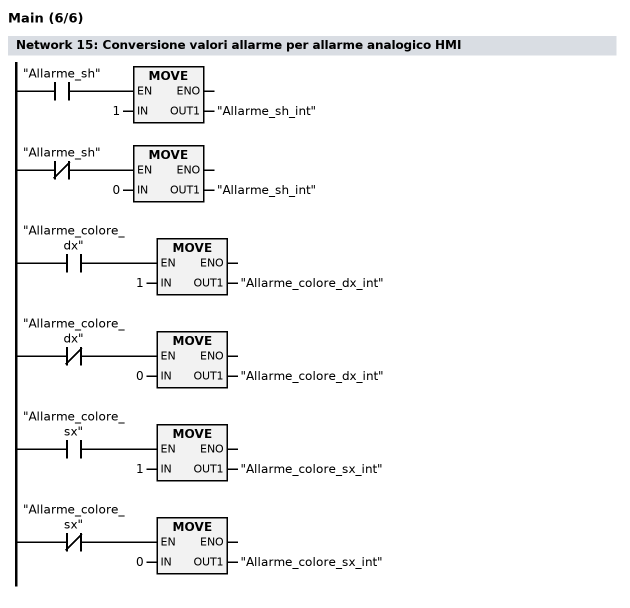
   RUNG wire#powerrail
      Contact( "Allarme_sh" )
      Move(in := 1, out1 => "Allarme_sh_int")
   END_RUNG
   RUNG wire#powerrail
      I_Contact( "Allarme_sh" )
      Move(in := 0, out1 => "Allarme_sh_int")
   END_RUNG
   RUNG wire#powerrail
      Contact( "Allarme_colore_dx" )
      Move(in := 1, out1 => "Allarme_colore_dx_int")
   END_RUNG
   RUNG wire#powerrail
      I_Contact( "Allarme_colore_dx" )
      Move(in := 0, out1 => "Allarme_colore_dx_int")
   END_RUNG
   RUNG wire#powerrail
      Contact( "Allarme_colore_sx" )
      Move(in := 1, out1 => "Allarme_colore_sx_int")
   END_RUNG
   RUNG wire#powerrail
      I_Contact( "Allarme_colore_sx" )
      Move(in := 0, out1 => "Allarme_colore_sx_int")
   END_RUNG
   // the same network as SCL:
   IF "Allarme_sh" THEN "Allarme_sh_int" := 1; END_IF;
   IF NOT "Allarme_sh" THEN "Allarme_sh_int" := 0; END_IF;
   IF "Allarme_colore_dx" THEN "Allarme_colore_dx_int" := 1; END_IF;
   IF NOT "Allarme_colore_dx" THEN "Allarme_colore_dx_int" := 0; END_IF;
   IF "Allarme_colore_sx" THEN "Allarme_colore_sx_int" := 1; END_IF;
   IF NOT "Allarme_colore_sx" THEN "Allarme_colore_sx_int" := 0; END_IF;
END_REGION
END_ORGANIZATION_BLOCK

(* ===== HMI "HMI_RT_1" =====
system functions are stored by id; their names below are inferred from use
connection "HMI_Connection_1": ETHERNET, SMART_S7_1200_OMS

HMI tags "Default tag table"
   "HMI_Robot" : Bool = PLC "Pick-place_DB".work AT %Q0.1, 1 s
   "HMI_ElevatorDx" : Bool = PLC Elevator_dx_DB.pronto_ricevere AT %I1.5, 1 s
   "HMI_ElevatorSx" : Bool = PLC Elevator_sx_DB.pronto_ricevere AT %I1.6, 1 s
   "HMI_Impianto" : Bool = PLC Impianto_attivo AT %M0.0, 1 s
   "HMI_Start" : Bool = PLC Cmd_start AT %M0.1, 1 s
   "HMI_Stop" : Bool = PLC Cmd_stop AT %M0.2, 1 s
   "HMI_Totali" : Int = PLC Pezzi_totali AT %MW10, 1 s
   "HMI_Blu" : Int = PLC Pezzi_blu AT %MW12, 1 s
   "HMI_Verdi" : Int = PLC Pezzi_verdi AT %MW14, 1 s
   "HMI_Grigi" : Int = PLC Pezzi_grigi AT %MW16, 1 s
   "HMI_Sospendi" : Bool = PLC Sospendi AT %M0.5, 1 s
   "HMI_Reset" : Bool = PLC Reset AT %M0.4, 1 s
   "HMI_Stato_sospeso" : Bool = PLC Supervisore_DB.Stato_sospeso AT %DB1.DBW0, 1 s
   "HMI_Stato_allarme_attivo" : Bool = PLC Allarme AT %M0.3, 1 s
   "Allarme_sh" : Bool = PLC Allarme_sh AT %M1.0, 1 s
   "Allarme_colore_sx" : Bool = PLC Allarme_colore_sx AT %M0.7, 1 s
   "Allarme_colore_dx" : Bool = PLC Allarme_colore_dx AT %M0.6, 1 s
   "HMI_Allarme_sh_int" : Int = PLC Allarme_sh_int AT %MW20, 1 s
   "HMI_Allarme_colore_dx_int" : Int = PLC Allarme_colore_dx_int AT %MW22, 1 s
   "HMI_Allarme_colore_sx_int" : Int = PLC Allarme_colore_sx_int AT %MW24, 1 s

analog alarms
   1: 'ALLARME: pezzo mancante dopo il robot', class Errors, trigger "HMI_Allarme_sh_int"
   2: 'ALLARME: colore non rilevato sul nastro destro', class Errors, trigger "HMI_Allarme_colore_dx_int"
   3: 'ALLARME: colore non rilevato sul nastro sinistro', class Errors, trigger "HMI_Allarme_colore_sx_int"

screen "Home" 800x480, template "Template_1"
   Button "HmiScreenItemData" at 7,42 size 173x59; TextOn 'Forzature'; TextOff 'Supervisione impianto'; PictureOn "Navigates to Forzature for KTP900 Basic+ PN 17.0.0.0"; PictureOff "Navigates to Forzature for KTP900 Basic+ PN 17.0.0.0"
      on Click: ActivateScreen("Supervisione impianto", 0)
   TextField "Text field_1" at 28,104 size 286x27; Text 'STATO GENERALE IMPIANTO'
   TextField "Text field_2" at 563,104 size 187x27; Text 'CONTEGGIO PEZZI'
   TextField "Text field_3" at 362,103 size 101x27; Text 'COMANDI'
   TextField "Text field_5" at 198,53 size 546x25; Text 'IMPIANTO DI PRODUZIONE E SMISTAMENTO AUTOMATIZZATO'
   TextField "Text field_6" at 562,158 size 68x25; Text 'TOTALI'
   TextField "Text field_7" at 568,215 size 40x25; Text 'BLU'
   TextField "Text field_8" at 562,269 size 59x25; Text 'VERDI'
   TextField "Text field_9" at 562,329 size 59x25; Text 'GRIGI'
   TextField "Text field_13" at 45,210 size 101x20; Text 'ROBOT PRONTO'
   TextField "Text field_15" at 21,268 size 177x20; Text 'ELEVATOR DESTRO PRONTO'
   TextField "Text field_14" at 19,332 size 187x20; Text 'ELEVATOR SINISTRO PRONTO'
   Circle "Circle_2" at 228,199 size 43x43
      Appearance <- "HMI_Robot"
   Circle "Circle_3" at 229,257 size 44x44
      Appearance <- "HMI_ElevatorDx"
   Circle "Circle_4" at 228,323 size 45x45
      Appearance <- "HMI_ElevatorSx"
   IOField "I/O field_1" at 654,154 size 96x32; FormatPattern s99999
      ProcessValue <- "HMI_Totali"
   IOField "I/O field_2" at 654,210 size 96x32; FormatPattern s99999
      ProcessValue <- "HMI_Blu"
   IOField "I/O field_3" at 656,266 size 96x32; FormatPattern s99999
      ProcessValue <- "HMI_Verdi"
   IOField "I/O field_4" at 654,329 size 96x32; FormatPattern s99999
      ProcessValue <- "HMI_Grigi"
   Button "Button_2" at 357,249 size 120x71; TextOff 'ARRESTO'
      on Release: ResetBit("HMI_Stop")
      on Press: SetBit("HMI_Stop")
   Button "Button_3" at 357,162 size 119x63; TextOff 'AVVIO'
      on Release: ResetBit("HMI_Start")
      on Press: SetBit("HMI_Start")
   TextField "Text field_4" at 50,154 size 119x20; Text 'IMPIANTO ATTIVO'
   Circle "Circle_1" at 226,141 size 42x42
      Appearance <- "HMI_Impianto"

screen "Supervisione impianto" 800x480, template "Template_1"
   TextField "HmiScreenItemData" at 157,55 size 505x33; Text 'Supervisione impianto'
   Button "Back" at 1,41 size 159x47; TextOn 'Back'; TextOff 'Home'
      on Click: ActivateScreen("Home", 0)
   Button "Button_1" at 54,139 size 163x69; TextOff 'SOSPENDI'
      on Press: SetBit("HMI_Sospendi")
      on Release: ResetBit("HMI_Sospendi")
   Button "Button_2" at 58,243 size 158x71; TextOff 'RESET'
      on Press: SetBit("HMI_Reset")
      on Release: ResetBit("HMI_Reset")
   TextField "Text field_1" at 260,157 size 165x27; Text 'STATO SOSPESO'
   Circle "Circle_1" at 471,145 size 48x48
      Appearance <- "HMI_Stato_sospeso"
   TextField "Text field_2" at 261,261 size 176x27; Text 'ALLARME ATTIVO'
   Circle "Circle_2" at 471,248 size 48x48
      Appearance <- "HMI_Stato_allarme_attivo"
   TextField "Text field_4" at 583,100 size 181x23; Text 'DETTAGLIO ALLARMI'
   TextField "Text field_5" at 572,139 size 193x20; Text 'Allarme mancata lavorazione'
   TextField "Text field_6" at 599,240 size 148x20; Text 'Allarme nastro destro'
   TextField "Text field_7" at 598,345 size 153x20; Text 'Allarme nastro sinistro'
   Circle "Circle_4" at 654,167 size 48x48
      Appearance <- "Allarme_sh"
   Circle "Circle_5" at 654,277 size 48x48
      Appearance <- "Allarme_colore_dx"
   Circle "Circle_6" at 654,376 size 48x48
      Appearance <- "Allarme_colore_sx"

Template "Template_1" 800x480
   Button "Exit" at 722,440 size 55x39; TextOn 'Exit'; TextOff 'Exit'; PictureOn "ExitRuntime_KTP900_Basic_PN_TR"; PictureOff "ExitRuntime_KTP900_Basic_PN_TR"
      on Release: StopRuntime(0)
   Button "Template_Button" at 622,440 size 55x39; TextOff 'Text'
   Button "Template_Button_1" at 522,440 size 55x39; TextOff 'Text'
   Button "Template_Button_2" at 422,440 size 55x39; TextOff 'Text'
   Button "Template_Button_3" at 322,440 size 55x39; TextOff 'Text'
   Button "Template_Button_4" at 222,440 size 55x39; TextOff 'Text'
   Button "Alarms" at 122,440 size 55x39; TextOn 'Alarms'; TextOff 'Alarms'; PictureOn "AlarmDisplay_KTP900_Basic_PN_TR"; PictureOff "AlarmDisplay_KTP900_Basic_PN_TR"
      on Release: function_ef3f5d25("Alarm window_Unacknowledged", -1)
   Button "Start screen" at 22,440 size 55x39; TextOn 'Start screen'; TextOff 'Start screen'; PictureOn "NavigateHome_KTP900_Basic_PN_TR"; PictureOff "NavigateHome_KTP900_Basic_PN_TR"
      on Release: ActivateScreen("Home", 0)
   SymbolicIOField "Symbolic_IO_Field_Screen" at 73,7 size 620x26; TextOn '1'; TextOff '0'; TextList "TextList_ScreenNames"
   DateTimeField "HmiScreenItemData" at 695,20 size 105x20
   DateTimeField "HmiScreenItemData_1" at 695,0 size 105x20
   GraphicView "Logo" at 0,0 size 71x40; Picture "Logo of HMI_1"
*)